(* IEC 61131-3 sources: conversion/test/strings, 10 files *)

(* ---- Asserts.st ---- *)
NAMESPACE AxUnit.Assert

    FUNCTION Equal
        VAR_INPUT
            expected : STRING;
            actual : STRING;
        END_VAR
        Equal(expected := TRUE, actual := expected = actual);
        ;
    END_FUNCTION

END_NAMESPACE

(* ---- ArrayToStringTest.st ---- *)
USING AxUnit.Assert;
USING System.Strings;

NAMESPACE Simatic.Ax.Conversion
    {TestFixture}
    CLASS ArrayToStringTest
        VAR PROTECTED
            array_1_10 : ARRAY[1..10] OF CHAR := ['1', '2', '3', '4', '5', '6', '7', '8', '9', '0'];
            array_0_9 : ARRAY[0..9] OF CHAR := ['0', '1', '2', '3', '4', '5', '6', '7', '8', '9'];
            exp_0_9 : STRING := '0123456789';
            exp_1_10 : STRING := '1234567890';
            empty_string : STRING;
            len : DINT;
            long_array : ARRAY[1..1024] OF CHAR;
            long_string : STRING := '12345678901234567890123456789012345678901234567890123456789012345678901234567890123456789012345678901234567890123456789012345678901234567890123456789012345678901234567890123456789012345678901234567890123456789012345678901234567890123456789012345678901234';
        END_VAR

        {Test}
        METHOD PUBLIC LongArrayTest_expect_StringLength_254
            VAR_TEMP
                _str : STRING;
            END_VAR            Strings.ToArray.OfCharCount(str := long_string, arr := long_array);
            // exceed string lenght
            long_array[255] := '5';
            long_array[256] := '6';
            long_array[257] := '7';

            _str := Arrays.ToString(arr := long_array);

            Equal(expected := 254, actual := LengthOf(_str));
            Equal(expected := long_string, actual := _str);

        END_METHOD

        {Test}
        METHOD PUBLIC Test_Array_ToString_End_smaller_than_start_expect_empty_string
            VAR_TEMP
                _str : STRING;
            END_VAR

            _str := Arrays.ToString(arr := array_0_9, startIdx := 9, endIdx := 5);
            Equal(expected := empty_string, actual := _str);
            ;
        END_METHOD

        {Test}
        METHOD PUBLIC Test_Array_ToString_without_indices_and_expect_full_string
            VAR_TEMP
                _str : STRING;
                array_0_9_test : string := '0123456789';
                array_1_10_test : string := '1234567890';
            END_VAR

            _str := Arrays.ToString(arr := array_0_9);
            Equal(expected := 10, actual := LengthOf(_str));
            Equal(expected := TRUE, actual := _str = array_0_9_test);

            _str := Arrays.ToString(arr := array_1_10);
            Equal(expected := 10, actual := LengthOf(_str));
            Equal(expected := TRUE, actual := _str = array_1_10_test);
            ;
        END_METHOD

        {Test}
        METHOD PUBLIC Test_Array_ToString_part_of_array_and_expect_correct_String
            VAR_TEMP
                _str : STRING;
            END_VAR

            _str := Arrays.ToString(arr := array_0_9, startIdx := 0, endIdx := 0);
            exp_0_9 := '0';
            Equal(expected := 1, actual := LengthOf(_str));
            Equal(expected := exp_0_9, actual := _str);

            _str := Arrays.ToString(arr := array_0_9, startIdx := 1, endIdx := 1);
            exp_0_9 := '1';
            Equal(expected := 1, actual := LengthOf(_str));
            Equal(expected := exp_0_9, actual := _str);

            _str := Arrays.ToString(arr := array_0_9, startIdx := 0, endIdx := 3);
            exp_0_9 := '0123';
            Equal(expected := 4, actual := LengthOf(_str));
            Equal(expected := exp_0_9, actual := _str);

            _str := Arrays.ToString(arr := array_0_9, startIdx := 1, endIdx := 5);
            exp_0_9 := '12345';
            Equal(expected := 5, actual := LengthOf(_str));
            Equal(expected := exp_0_9, actual := _str);

            _str := Arrays.ToString(arr := array_1_10, startIdx := 1, endIdx := 5);
            exp_1_10 := '23456';
            Equal(expected := 5, actual := LengthOf(_str));
            Equal(expected := exp_1_10, actual := _str);
            ;
        END_METHOD

        {Test}
        METHOD PUBLIC Test_Array_Invalid_Indices_Expect_empty_Strings
            VAR_TEMP
                _str : STRING;
            END_VAR

            _str := Arrays.ToString(arr := array_1_10, startIdx := 0, endIdx := 11);
            exp_0_9 := '';
            Equal(expected := 0, actual := LengthOf(_str));
            Equal(expected := exp_0_9, actual := _str);
            ;
            _str := Arrays.ToString(arr := array_1_10, startIdx := 0, endIdx := 10);
            exp_0_9 := '';
            Equal(expected := 0, actual := LengthOf(_str));
            Equal(expected := exp_0_9, actual := _str);

            _str := Arrays.ToString(arr := array_1_10, startIdx := -1, endIdx := 10);
            exp_0_9 := '';
            Equal(expected := 0, actual := LengthOf(_str));
            Equal(expected := exp_0_9, actual := _str);
            ;
        END_METHOD
    END_CLASS
END_NAMESPACE

(* ---- StringToAnyTest.st ---- *)
USING AxUnit.Assert;
USING System.Strings;

NAMESPACE Simatic.Ax.Conversion
    {TestFixture}
    CLASS StrinToAnyIntTest
        VAR
            val : LINT;
            val2 : ULINT;
            res : BOOL;
        END_VAR

        {Test}
        METHOD PUBLIC Convert_STRING_0_TO_LINT_0
            res := StringToAnyInt(str := '0', value => val);
            Equal(expected := 0, actual := val);
            Equal(expected := TRUE, actual := res);
        END_METHOD

        {Test}
        METHOD PUBLIC Convert_STRING_0000000000000000_TO_LINT_0
            res := StringToAnyInt(str := '0000000000000000', value => val);
            Equal(expected := 0, actual := val);
            Equal(expected := TRUE, actual := res);
        END_METHOD

        //ToDo after bugfix
        // {Test(str := STRING#'', value := ULINT#0, success :=FALSE)}
        // {Test(str := STRING#'+', value := ULINT#0, success :=FALSE)}
        // {Test(str := STRING#'-', value := ULINT#0, success :=FALSE)}
        // {Test(str := STRING#'0', value := ULINT#0, success :=TRUE)}
        // {Test(str := STRING#'1', value := ULINT#1, success :=TRUE)}
        // {Test(str := STRING#'2', value := ULINT#2, success :=TRUE)}
        // {Test(str := STRING#'3', value := ULINT#3, success :=TRUE)}
        // {Test(str := STRING#'4', value := ULINT#4, success :=TRUE)}
        // {Test(str := STRING#'5', value := ULINT#5, success :=TRUE)}
        // {Test(str := STRING#'6', value := ULINT#6, success :=TRUE)}
        // {Test(str := STRING#'7', value := ULINT#7, success :=TRUE)}
        // {Test(str := STRING#'8', value := ULINT#8, success :=TRUE)}
        // {Test(str := STRING#'9', value := ULINT#9, success :=TRUE)}
        // {Test(str := STRING#'10', value := ULINT#10, success :=TRUE)}
        // {Test(str := STRING#'15', value := ULINT#15, success :=TRUE)}
        // {Test(str := STRING#'18446744073709551600', value := ULINT#18446744073709551600, success :=TRUE)}
        // {Test(str := STRING#'18446744073709551601', value := ULINT#18446744073709551601, success :=TRUE)}
        // {Test(str := STRING#'18446744073709551602', value := ULINT#18446744073709551602, success :=TRUE)}
        // {Test(str := STRING#'18446744073709551603', value := ULINT#18446744073709551603, success :=TRUE)}
        // {Test(str := STRING#'18446744073709551604', value := ULINT#18446744073709551604, success :=TRUE)}
        // {Test(str := STRING#'18446744073709551605', value := ULINT#18446744073709551605, success :=TRUE)}
        // {Test(str := STRING#'18446744073709551606', value := ULINT#18446744073709551606, success :=TRUE)}
        // {Test(str := STRING#'18446744073709551607', value := ULINT#18446744073709551607, success :=TRUE)}
        // {Test(str := STRING#'18446744073709551608', value := ULINT#18446744073709551608, success :=TRUE)}
        // {Test(str := STRING#'18446744073709551609', value := ULINT#18446744073709551609, success :=TRUE)}
        // {Test(str := STRING#'18446744073709551610', value := ULINT#18446744073709551610, success :=TRUE)}
        // {Test(str := STRING#'18446744073709551611', value := ULINT#18446744073709551611, success :=TRUE)}
        // {Test(str := STRING#'18446744073709551612', value := ULINT#18446744073709551612, success :=TRUE)}
        // {Test(str := STRING#'18446744073709551613', value := ULINT#18446744073709551613, success :=TRUE)}
        // {Test(str := STRING#'18446744073709551614', value := ULINT#18446744073709551614, success :=TRUE)}
        // {Test(str := STRING#'18446744073709551615', value := ULINT#18446744073709551615, success :=TRUE)}
        // {Test(str := STRING#'18446744073709551616', value := ULINT#0, success :=FALSE)}
        // {Test(str := STRING#'18446744073709551617', value := ULINT#0, success :=FALSE)}
        // {Test(str := STRING#'18446744073709551618', value := ULINT#0, success :=FALSE)}
        // {Test(str := STRING#'18446744073709551619', value := ULINT#0, success :=FALSE)}
        // {Test(str := STRING#'18446744073709551620', value := ULINT#0, success :=FALSE)}
        // {Test(str := STRING#'18446744073709551621', value := ULINT#0, success :=FALSE)}
        // {Test(str := STRING#'18446744073709551622', value := ULINT#0, success :=FALSE)}
        // {Test(str := STRING#'18446744073709551623', value := ULINT#0, success :=FALSE)}
        // {Test(str := STRING#'18446744073709551624', value := ULINT#0, success :=FALSE)}
        // {Test(str := STRING#'18446744073709551625', value := ULINT#0, success :=FALSE)}
        // {Test(str := STRING#'18446744073709551626', value := ULINT#0, success :=FALSE)}
        // {Test(str := STRING#'18446744073709551636', value := ULINT#0, success :=FALSE)}
        // {Test(str := STRING#'18446744073709551746', value := ULINT#0, success :=FALSE)}
        // {Test(str := STRING#'18446744073709551800', value := ULINT#0, success :=FALSE)}
        // {Test(str := STRING#'20000000000000000000', value := ULINT#0, success :=FALSE)}
        // METHOD PUBLIC Convert_STRING_TO_ULINT
        //     VAR_INPUT
        //         str : STRING;
        //         value : ULINT;
        //         success : BOOL;
        //     END_VAR
        //     VAR_TEMP
        //         resVal : ULINT;
        //     END_VAR
        //     res := StringToULint(str := str, value => resVal);
        //     Equal(expected := value, actual := resVal);
        //     Equal(expected := success, actual := res);
        // END_METHOD

        // {Test(str := STRING#'', value := LINT#0, success :=FALSE)}
        // {Test(str := STRING#'+', value := LINT#0, success :=FALSE)}
        // {Test(str := STRING#'-', value := LINT#0, success :=FALSE)}
        // {Test(str := STRING#'0', value := LINT#0, success :=TRUE)}
        // {Test(str := STRING#'1', value := LINT#1, success :=TRUE)}
        // {Test(str := STRING#'2', value := LINT#2, success :=TRUE)}
        // {Test(str := STRING#'3', value := LINT#3, success :=TRUE)}
        // {Test(str := STRING#'4', value := LINT#4, success :=TRUE)}
        // {Test(str := STRING#'5', value := LINT#5, success :=TRUE)}
        // {Test(str := STRING#'6', value := LINT#6, success :=TRUE)}
        // {Test(str := STRING#'7', value := LINT#7, success :=TRUE)}
        // {Test(str := STRING#'8', value := LINT#8, success :=TRUE)}
        // {Test(str := STRING#'9', value := LINT#9, success :=TRUE)}
        // {Test(str := STRING#'10', value := LINT#10, success :=TRUE)}
        // {Test(str := STRING#'15', value := LINT#15, success :=TRUE)}
        // {Test(str := STRING#'-0', value := LINT#0, success :=TRUE)}
        // {Test(str := STRING#'-1', value := LINT#-1, success :=TRUE)}
        // {Test(str := STRING#'-2', value := LINT#-2, success :=TRUE)}
        // {Test(str := STRING#'-3', value := LINT#-3, success :=TRUE)}
        // {Test(str := STRING#'-4', value := LINT#-4, success :=TRUE)}
        // {Test(str := STRING#'-5', value := LINT#-5, success :=TRUE)}
        // {Test(str := STRING#'-6', value := LINT#-6, success :=TRUE)}
        // {Test(str := STRING#'-7', value := LINT#-7, success :=TRUE)}
        // {Test(str := STRING#'-8', value := LINT#-8, success :=TRUE)}
        // {Test(str := STRING#'-9', value := LINT#-9, success :=TRUE)}
        // {Test(str := STRING#'-10', value := LINT#-10, success :=TRUE)}
        // {Test(str := STRING#'-15', value := LINT#-15, success :=TRUE)}
        // {Test(str := STRING#'9223372036854775799', value := LINT#9223372036854775799, success :=TRUE)}
        // {Test(str := STRING#'9223372036854775800', value := LINT#9223372036854775800, success :=TRUE)}
        // {Test(str := STRING#'9223372036854775801', value := LINT#9223372036854775801, success :=TRUE)}
        // {Test(str := STRING#'9223372036854775802', value := LINT#9223372036854775802, success :=TRUE)}
        // {Test(str := STRING#'9223372036854775803', value := LINT#9223372036854775803, success :=TRUE)}
        // {Test(str := STRING#'9223372036854775804', value := LINT#9223372036854775804, success :=TRUE)}
        // {Test(str := STRING#'9223372036854775805', value := LINT#9223372036854775805, success :=TRUE)}
        // {Test(str := STRING#'9223372036854775806', value := LINT#9223372036854775806, success :=TRUE)}
        // {Test(str := STRING#'9223372036854775807', value := LINT#9223372036854775807, success :=TRUE)}
        // {Test(str := STRING#'9223372036854775808', value := LINT#0, success :=FALSE)}
        // {Test(str := STRING#'9223372036854775809', value := LINT#0, success :=FALSE)}
        // {Test(str := STRING#'9223372036854775810', value := LINT#0, success :=FALSE)}
        // {Test(str := STRING#'9223372036854775811', value := LINT#0, success :=FALSE)}
        // {Test(str := STRING#'19223372036854775811', value := LINT#0, success :=FALSE)}

        // {Test(str := STRING#'-9223372036854775799', value := LINT#-9223372036854775799, success :=TRUE)}
        // {Test(str := STRING#'-9223372036854775800', value := LINT#-9223372036854775800, success :=TRUE)}
        // {Test(str := STRING#'-9223372036854775801', value := LINT#-9223372036854775801, success :=TRUE)}
        // {Test(str := STRING#'-9223372036854775802', value := LINT#-9223372036854775802, success :=TRUE)}
        // {Test(str := STRING#'-9223372036854775803', value := LINT#-9223372036854775803, success :=TRUE)}
        // {Test(str := STRING#'-9223372036854775804', value := LINT#-9223372036854775804, success :=TRUE)}
        // {Test(str := STRING#'-9223372036854775805', value := LINT#-9223372036854775805, success :=TRUE)}
        // {Test(str := STRING#'-9223372036854775806', value := LINT#-9223372036854775806, success :=TRUE)}
        // {Test(str := STRING#'-9223372036854775807', value := LINT#-9223372036854775807, success :=TRUE)}
        // {Test(str := STRING#'-9223372036854775808', value := LINT#-9223372036854775808, success :=TRUE)}
        // {Test(str := STRING#'-9223372036854775809', value := LINT#0, success :=FALSE)}
        // {Test(str := STRING#'-9223372036854775810', value := LINT#0, success :=FALSE)}
        // {Test(str := STRING#'-9223372036854775811', value := LINT#0, success :=FALSE)}
        // {Test(str := STRING#'-19223372036854775811', value := LINT#0, success :=FALSE)}
        // METHOD PUBLIC Convert_STRING_TO_ANYINT
        //     VAR_INPUT
        //         str : STRING;
        //         value : LINT;
        //         success : BOOL;
        //     END_VAR
        //     VAR_TEMP
        //         resVal : LINT;
        //     END_VAR
        //     res := StringToAnyInt(str := str, value => resVal);
        //     Equal(expected := value, actual := resVal);
        //     Equal(expected := success, actual := res);
        // END_METHOD

        {Test}
        METHOD PUBLIC Convert_STRING_123_TO_LINT_123
            res := StringToAnyInt(str := '123', value => val);
            Equal(expected := 123, actual := val);
            Equal(expected := TRUE, actual := res);
        END_METHOD

        {Test}
        METHOD PUBLIC Convert_STRING_00000000123_TO_LINT_123
            res := StringToAnyInt(str := '123', value => val);
            Equal(expected := 123, actual := val);
            Equal(expected := TRUE, actual := res);
        END_METHOD

        {Test}
        METHOD PUBLIC Convert_STRING_PLUS_123_TO_LINT_123
            res := StringToAnyInt(str := '+00000000123', value => val);
            Equal(expected := 123, actual := val);
            Equal(expected := TRUE, actual := res);
        END_METHOD

        {Test}
        METHOD PUBLIC Convert_STRING_MINUS_0000000000123_TO_LINT_123
            res := StringToAnyInt(str := '-00000000123', value => val);
            Equal(expected := -123, actual := val);
            Equal(expected := TRUE, actual := res);
        END_METHOD

        {Test}
        METHOD PUBLIC Convert_STRING_MINUS_123_TO_LINT_123
            res := StringToAnyInt(str := '-123', value => val);
            Equal(expected := -123, actual := val);
            Equal(expected := TRUE, actual := res);
        END_METHOD

        {Test}
        METHOD PUBLIC Convert_STRING_MINUS_1234567890_TO_LINT_1234567890
            res := StringToAnyInt(str := '-1234567890', value => val);
            Equal(expected := LINT#-1234567890, actual := val);
            Equal(expected := TRUE, actual := res);
        END_METHOD

        {Test}
        METHOD PUBLIC Convert_STRING_9223372036854775807_TO_LINT_9223372036854775807
            res := StringToAnyInt(str := '9223372036854775807', value => val);
            Equal(expected := LINT#9223372036854775807, actual := val);
            Equal(expected := TRUE, actual := res);
            res := StringToAnyInt(str := '+9223372036854775807', value => val);
            Equal(expected := LINT#9223372036854775807, actual := val);
            Equal(expected := TRUE, actual := res);

        END_METHOD

        {Test}
        METHOD PUBLIC Convert_STRING_MINUS_9223372036854775808_TO_LINT_9223372036854775808
            res := StringToAnyInt(str := '-9223372036854775808', value => val);
            Equal(expected := LINT#-9223372036854775808, actual := val);
            Equal(expected := TRUE, actual := res);
        END_METHOD

        {Test}
        METHOD PUBLIC Convert_STRING_18446744073709551615_TO_ULINT_18446744073709551615
            res := StringToULINT(str := '18446744073709551615', value => val2);
            Equal(expected := ULINT#18446744073709551615, actual := val2);
            Equal(expected := TRUE, actual := res);

            res := StringToULINT(str := '+18446744073709551615', value => val2);
            Equal(expected := ULINT#18446744073709551615, actual := val2);
            Equal(expected := TRUE, actual := res);
        END_METHOD

        {Test}
        METHOD PUBLIC Convert_WrongStrings_ExpectFalse
            res := StringToAnyInt(str := '+-123', value => val);
            Equal(expected := 0, actual := val);
            Equal(expected := FALSE, actual := res);

            res := StringToAnyInt(str := '000+123', value => val);
            Equal(expected := 0, actual := val);
            Equal(expected := FALSE, actual := res);

            res := StringToAnyInt(str := '1000+123', value => val);
            Equal(expected := 0, actual := val);
            Equal(expected := FALSE, actual := res);

            res := StringToAnyInt(str := 'aaa', value => val);
            Equal(expected := 0, actual := val);
            Equal(expected := FALSE, actual := res);

            res := StringToAnyInt(str := '12a23', value => val);
            Equal(expected := 0, actual := val);
            Equal(expected := FALSE, actual := res);

        END_METHOD
    END_CLASS
END_NAMESPACE

(* ---- StringToArrayOfLintCountTest.st ---- *)
USING AxUnit.Assert;
USING System.Strings;

NAMESPACE Simatic.Ax.Conversion.Strings.ToArray
    {TestFixture}
    CLASS StringToArrayOfLIntCountTest
        VAR
            arr: ARRAY[0..3] OF LINT;
        END_VAR

        {Test}
        METHOD PUBLIC EmptyArray_ReturnsFalse
            VAR
                str: STRING := '';
                count: DINT;
            END_VAR

            count := ToArray.OfLintCount(str, arr);
            Equal(0, count);

            str:= '   ';
            count := ToArray.OfLintCount(str, arr);
            Equal(0, count);
        END_METHOD

        {Test}
        METHOD PUBLIC NotArray_ReturnsFalse
            VAR
                str: STRING := 'hello';
                count: DINT;
            END_VAR
            count := ToArray.OfLintCount(str, arr);
            Equal(0, count);
        END_METHOD

        {Test}
        METHOD PUBLIC WrongArray_ReturnsFalse
            VAR
                str: STRING := '["hello", "goodbye"]';
                count: DINT;
            END_VAR
            count := ToArray.OfLintCount(str, arr);
            Equal(0, count);
        END_METHOD

        {Test}
        METHOD PUBLIC Array_Converts
            VAR
                str: STRING := '[12, 345, 6789, 101112]';
                count: DINT;
            END_VAR
            count := ToArray.OfLintCount(str, arr);
            Equal(4, count);
            Equal(LINT#12, arr[0]);
            Equal(LINT#345, arr[1]);
            Equal(LINT#6789, arr[2]);
            Equal(LINT#101112, arr[3]);
        END_METHOD

        {Test}
        METHOD PUBLIC Array_Converts_with_spaces
            VAR
                str: STRING := '   [   12,   345   ,    6789    ,    101112    ]   ';
                count: DINT;
            END_VAR
            count := ToArray.OfLintCount(str, arr);
            Equal(4, count);
            Equal(LINT#12, arr[0]);
            Equal(LINT#345, arr[1]);
            Equal(LINT#6789, arr[2]);
            Equal(LINT#101112, arr[3]);
        END_METHOD

        {Test}
        METHOD PUBLIC Smaller_Array_Converts_with_spaces
            VAR
                str: STRING := '   [   345   ,    6789    ,    101112    ]   ';
                count: DINT;
            END_VAR
            count := ToArray.OfLintCount(str, arr);
            Equal(3, count);
            Equal(LINT#345, arr[0]);
            Equal(LINT#6789, arr[1]);
            Equal(LINT#101112, arr[2]);
        END_METHOD

        {Test}
        METHOD PUBLIC Array_Converts_toSmallArray
            VAR
                str: STRING := '[12, 345, 6789, 101112, 1234]';
                count: DINT;
            END_VAR
            count := ToArray.OfLintCount(str, arr);
            Equal(4, count);
            Equal(LINT#12, arr[0]);
            Equal(LINT#345, arr[1]);
            Equal(LINT#6789, arr[2]);
            Equal(LINT#101112, arr[3]);
        END_METHOD

        {Test}
        METHOD PUBLIC Array_Converts_toBigArray
            VAR
                str: STRING := '[12, 345, 6789]';
                count: DINT;
            END_VAR
            count := ToArray.OfLintCount(str, arr);
            Equal(3, count);
            Equal(LINT#12, arr[0]);
            Equal(LINT#345, arr[1]);
            Equal(LINT#6789, arr[2]);
        END_METHOD

    END_CLASS
END_NAMESPACE

(* ---- StringToArrayTest.st ---- *)
USING AxUnit.Assert;
USING System.Strings;

NAMESPACE Simatic.Ax.Conversion
    {TestFixture}
    CLASS StrinToArrayIntTest
        VAR PROTECTED
            s10 : STRING := '0123456789';
            s16 : STRING := '0123456789ABCDEF';
            a0_9 : ARRAY[0..9] OF CHAR;
            a10_19 : ARRAY[10..19] OF CHAR;

            a0_12 : ARRAY[0..12] OF CHAR;
            a10_22 : ARRAY[10..12] OF CHAR;
            len : DINT;
        END_VAR

        {Test}
        METHOD PUBLIC Test_array_and_string_length_is_equal_expect_lenght_10
            len := Strings.ToArray.OfCharCount(s10, a0_9);
            Equal(expected := 10, actual := len);
            Equal(expected := '0', actual := a0_9[0]);
            Equal(expected := '1', actual := a0_9[1]);
            Equal(expected := '8', actual := a0_9[8]);
            Equal(expected := '9', actual := a0_9[9]);
        END_METHOD

        {Test}
        METHOD PUBLIC Test_array_starting_with_10_and_string_length_is_equal_expect_lenght_10
            len := Strings.ToArray.OfCharCount(s10, a10_19);
            Equal(expected := 10, actual := len);
            Equal(expected := '0', actual := a10_19[10]);
            Equal(expected := '1', actual := a10_19[11]);
            Equal(expected := '8', actual := a10_19[18]);
            Equal(expected := '9', actual := a10_19[19]);
        END_METHOD

        {Test}
        METHOD PUBLIC Test_array_and_string_length_is_longer_expect_lenght_10
            len := Strings.ToArray.OfCharCount(s16, a0_9);
            Equal(expected := 10, actual := len);
            Equal(expected := '0', actual := a0_9[0]);
            Equal(expected := '1', actual := a0_9[1]);
            Equal(expected := '8', actual := a0_9[8]);
            Equal(expected := '9', actual := a0_9[9]);
        END_METHOD

        {Test}
        METHOD PUBLIC Test_array_starting_with_10_and_string_length_is_longer_expect_lenght_10
            len := Strings.ToArray.OfCharCount(s16, a10_19);
            Equal(expected := 10, actual := len);
            Equal(expected := '0', actual := a10_19[10]);
            Equal(expected := '1', actual := a10_19[11]);
            Equal(expected := '8', actual := a10_19[18]);
            Equal(expected := '9', actual := a10_19[19]);
        END_METHOD

        {Test}
        METHOD PUBLIC Test_array_and_string_length_buffer_is_longer_expect_lenght_10
            len := Strings.ToArray.OfCharCount(s10, a0_12);
            Equal(expected := 10, actual := len);
            Equal(expected := '0', actual := a0_12[0]);
            Equal(expected := '1', actual := a0_12[1]);
            Equal(expected := '8', actual := a0_12[8]);
            Equal(expected := '9', actual := a0_12[9]);
            Equal(expected := TO_CHAR(BYTE#0), actual := a0_12[10]);
            Equal(expected := TO_CHAR(BYTE#0), actual := a0_12[11]);
            Equal(expected := TO_CHAR(BYTE#0), actual := a0_12[12]);

            len := Strings.ToArray.OfCharCount(s16, a0_12);
            Equal(expected := 13, actual := len);
        END_METHOD

        {Test}
        METHOD PUBLIC Test_array_and_string_length_buffer_is_shorter_expect_lenght_13

            len := Strings.ToArray.OfCharCount(s16, a0_12);
            Equal(expected := 13, actual := len);
            Equal(expected := '0', actual := a0_12[0]);
            Equal(expected := '1', actual := a0_12[1]);
            Equal(expected := '8', actual := a0_12[8]);
            Equal(expected := '9', actual := a0_12[9]);
            Equal(expected := 'A', actual := a0_12[10]);
            Equal(expected := 'B', actual := a0_12[11]);
            Equal(expected := 'C', actual := a0_12[12]);
        END_METHOD
    END_CLASS
END_NAMESPACE

(* ---- TestDifferentTypeConversions.st ---- *)
USING AxUnit.Assert;
using System.Strings;

NAMESPACE Simatic.Ax.Conversion
    {TestFixture}
    CLASS TestDifferentTypeConversions
        {Test}
        METHOD PUBLIC Test_SINT
            Equal(expected := '0', actual := Integer.ToString(value := SINT#0));
            Equal(expected := '127', actual := Integer.ToString(value := SINT#127));
            Equal(expected := '+127', actual := Integer.ToString(value := USINT#127, mode := ConversionMode#FORCE_SIGN));
            Equal(expected := '-128', actual := Integer.ToString(value := SINT#-128));
        END_METHOD

        {Test}
        METHOD PUBLIC Test_USINT
            Equal(expected := '0', actual := Integer.ToString(value := USINT#0));
            Equal(expected := '255', actual := Integer.ToString(value := USINT#255));
            Equal(expected := '+255', actual := Integer.ToString(value := USINT#255, mode := ConversionMode#FORCE_SIGN));
        END_METHOD

        {Test}
        METHOD PUBLIC Test_INT
            Equal(expected := '0', actual := Integer.ToString(value := INT#0));
            Equal(expected := '32767', actual := Integer.ToString(value := INT#32767));
            Equal(expected := '+32767', actual := Integer.ToString(value := INT#32767, mode := ConversionMode#FORCE_SIGN));
            Equal(expected := '-32768', actual := Integer.ToString(value := INT#-32768));

        END_METHOD

        {Test}
        METHOD PUBLIC Test_UINT
            Equal(expected := '0', actual := Integer.ToString(value := UINT#0));
            Equal(expected := '65535', actual := Integer.ToString(value := UINT#65535));
            Equal(expected := '+65535', actual := Integer.ToString(value := UINT#65535, mode := ConversionMode#FORCE_SIGN));

        END_METHOD

        {Test}
        METHOD PUBLIC Test_DINT
            Equal(expected := '0', actual := Integer.ToString(value := DINT#0));
            Equal(expected := '2147483647', actual := Integer.ToString(value := DINT#2147483647));
            Equal(expected := '+2147483647', actual := Integer.ToString(value := UDINT#2147483647, mode := ConversionMode#FORCE_SIGN));
            Equal(expected := '-2147483648', actual := Integer.ToString(value := DINT#-2147483648));
        END_METHOD

        {Test}
        METHOD PUBLIC Test_UDINT
            Equal(expected := '0', actual := Integer.ToString(value := UDINT#0));
            Equal(expected := '+4294967295', actual := Integer.ToString(value := UDINT#4294967295, mode := ConversionMode#FORCE_SIGN));
            Equal(expected := '4294967295', actual := Integer.ToString(value := UDINT#4294967295));
        END_METHOD

        {Test}
        METHOD PUBLIC Test_LINT
            Equal(expected := '0', actual := Integer.ToString(value := DINT#0));
            Equal(expected := '9223372036854775807', actual := Integer.ToString(value := LINT#9223372036854775807));
            Equal(expected := '+9223372036854775807', actual := Integer.ToString(value := LINT#9223372036854775807, mode := ConversionMode#FORCE_SIGN));
            Equal(expected := '-9223372036854775808', actual := Integer.ToString(value := LINT#-9223372036854775808));
        END_METHOD

        {Test}
        METHOD PUBLIC Test_ULINT
            Equal(expected := '0', actual := Integer.ToString(value := UDINT#0));
            Equal(expected := '18446744073709551615', actual := Integer.ToString(value := ULINT#18446744073709551615));
            Equal(expected := '+18446744073709551615', actual := Integer.ToString(value := ULINT#18446744073709551615, mode := ConversionMode#FORCE_SIGN));

        END_METHOD

    END_CLASS
END_NAMESPACE

(* ---- TestGetHexValueOfChar.st ---- *)
USING AxUnit.Assert;
NAMESPACE Simatic.Ax.Conversion
    {TestFixture}
    CLASS TestGetHexValueOfChar
        VAR PROTECTED
            res : BYTE;
            ret : bool;
        END_VAR

        {Test(c := 'a', n := 1, exp := BYTE#16#a)}
        {Test(c := 'b', n := 1, exp := BYTE#16#b)}
        {Test(c := 'c', n := 1, exp := BYTE#16#c)}
        {Test(c := 'd', n := 1, exp := BYTE#16#d)}
        {Test(c := 'e', n := 1, exp := BYTE#16#e)}
        {Test(c := 'f', n := 1, exp := BYTE#16#f)}
        {Test(c := 'A', n := 1, exp := BYTE#16#a)}
        {Test(c := 'B', n := 1, exp := BYTE#16#b)}
        {Test(c := 'C', n := 1, exp := BYTE#16#c)}
        {Test(c := 'D', n := 1, exp := BYTE#16#d)}
        {Test(c := 'E', n := 1, exp := BYTE#16#e)}
        {Test(c := 'F', n := 1, exp := BYTE#16#f)}
        {Test(c := '0', n := 1, exp := BYTE#16#0)}
        {Test(c := '1', n := 1, exp := BYTE#16#1)}
        {Test(c := '2', n := 1, exp := BYTE#16#2)}
        {Test(c := '3', n := 1, exp := BYTE#16#3)}
        {Test(c := '4', n := 1, exp := BYTE#16#4)}
        {Test(c := '5', n := 1, exp := BYTE#16#5)}
        {Test(c := '6', n := 1, exp := BYTE#16#6)}
        {Test(c := '7', n := 1, exp := BYTE#16#7)}
        {Test(c := '8', n := 1, exp := BYTE#16#8)}
        {Test(c := '9', n := 1, exp := BYTE#16#9)}
        METHOD PUBLIC ConvertHexCharsToByteValue
            VAR_INPUT
                c : CHAR;
                n : INT;
                exp : BYTE;
            END_VAR
            ret := GetHexValueOfChar(c := c, result => res);
            Equal(expected := exp, actual := res);
            Equal(expected := TRUE, actual := ret);
            ;
        END_METHOD

        {Test}
        METHOD PUBLIC InvalidCharacter
            ret := GetHexValueOfChar(c := 'h', result => res);
            Equal(expected := FALSE, actual := ret);
        END_METHOD
    END_CLASS
END_NAMESPACE

(* ---- TestStringToHex.st ---- *)
USING AxUnit.Assert;
NAMESPACE Simatic.Ax.Conversion.Strings
    {TestFixture}
    CLASS TestStringToHex
        VAR PROTECTED
            res : DWORD;
            ret : WORD;
        END_VAR

        //ToDo after bugfix
        // {Test(str := 'a', n := 1, exp := DWORD#16#a)}
        // {Test(str := 'b', n := 1, exp := DWORD#16#b)}
        // {Test(str := 'c', n := 1, exp := DWORD#16#c)}
        // {Test(str := 'd', n := 1, exp := DWORD#16#d)}
        // {Test(str := 'e', n := 1, exp := DWORD#16#e)}
        // {Test(str := 'f', n := 1, exp := DWORD#16#f)}
        // {Test(str := 'A', n := 1, exp := DWORD#16#a)}
        // {Test(str := 'B', n := 1, exp := DWORD#16#b)}
        // {Test(str := 'C', n := 1, exp := DWORD#16#c)}
        // {Test(str := 'D', n := 1, exp := DWORD#16#d)}
        // {Test(str := 'E', n := 1, exp := DWORD#16#e)}
        // {Test(str := 'F', n := 1, exp := DWORD#16#f)}
        // {Test(str := '0', n := 1, exp := DWORD#16#0)}
        // {Test(str := '1', n := 1, exp := DWORD#16#1)}
        // {Test(str := '2', n := 1, exp := DWORD#16#2)}
        // {Test(str := '3', n := 1, exp := DWORD#16#3)}
        // {Test(str := '4', n := 1, exp := DWORD#16#4)}
        // {Test(str := '5', n := 1, exp := DWORD#16#5)}
        // {Test(str := '6', n := 1, exp := DWORD#16#6)}
        // {Test(str := '7', n := 1, exp := DWORD#16#7)}
        // {Test(str := '8', n := 1, exp := DWORD#16#8)}
        // {Test(str := '9', n := 1, exp := DWORD#16#9)}
        // {Test(str := 'aFFe', n := 4, exp := DWORD#16#affe)}
        // {Test(str := 'aa', n := 2, exp := DWORD#16#aa)}
        // {Test(str := '12', n := 2, exp := DWORD#16#12)}
        // {Test(str := '123', n := 3, exp := DWORD#16#123)}
        // {Test(str := '1234', n := 4, exp := DWORD#16#1234)}
        // METHOD PUBLIC ConvertDifferentValidStringsToDWORD
        //     VAR_INPUT
        //         str : STRING;
        //         n : INT;
        //         exp : DWORD;
        //     END_VAR
        //     ret := ToHex(str := str, n := n, result => res);
        //     Equal(expected := exp, actual := res);
        //     Equal(expected := WORD#16#0000, actual := ret);
        //     ;
        // END_METHOD

        {Test}
        METHOD PUBLIC InvalidCharacter
            ret := ToHex(str := 'afgh', n := 4, result => res);
            Equal(expected := WORD#16#0007, actual := ret);
        END_METHOD

        {Test}
        METHOD PUBLIC InputSmallerThanN
            ret := ToHex(str := 'af', n := 3, result => res);
            Equal(expected := WORD#16#8182, actual := ret);
        END_METHOD

        {Test}
        METHOD PUBLIC OutputBufferToSmall
            ret := ToHex(str := '1234567890', n := 10, result => res);
            Equal(expected := WORD#16#8482, actual := ret);
        END_METHOD
    END_CLASS
END_NAMESPACE

(* ---- ToStringTest.st ---- *)
USING AxUnit.Assert;
USING System.Strings;

NAMESPACE Simatic.Ax.Conversion
    {TestFixture}
    CLASS ToStringTest
        VAR
            s : STRING;
        END_VAR
        {Test}
        METHOD PUBLIC Convert_INT_1234_ToString_Expect_1234
            s := AnyIntToString(value := 1234);
            Equal(expected := '1234', actual := s);
            Equal(expected := 4, actual := LengthOf(s));
        END_METHOD

        {Test}
        METHOD PUBLIC Convert_INT_MINUS_1234_ToString_Expect_MINUS_1234
            s := AnyIntToString(value := -1234);
            Equal(expected := '-1234', actual := s);
            Equal(expected := 5, actual := LengthOf(s));
        END_METHOD

        {Test}
        METHOD PUBLIC Convert_INT_VALUES_ToString_Expect_Value_AsString
            // 0
            s := AnyIntToString(value := 0);
            Equal(expected := '0', actual := s);
            Equal(expected := 1, actual := LengthOf(s));

            // 1
            s := AnyIntToString(value := 1);
            Equal(expected := '1', actual := s);
            Equal(expected := 1, actual := LengthOf(s));

            // 1
            s := AnyIntToString(value := -1);
            Equal(expected := '-1', actual := s);
            Equal(expected := 2, actual := LengthOf(s));

            // 99
            s := AnyIntToString(value := 99);
            Equal(expected := '99', actual := s);
            Equal(expected := 2, actual := LengthOf(s));

            // -99
            s := AnyIntToString(value := -99);
            Equal(expected := '-99', actual := s);
            Equal(expected := 3, actual := LengthOf(s));

            // 1234567890
            s := AnyIntToString(value := DINT#1234567890);
            Equal(expected := '1234567890', actual := s);
            Equal(expected := 10, actual := LengthOf(s));

            // -1234567890
            s := AnyIntToString(value := DINT#-1234567890);
            Equal(expected := '-1234567890', actual := s);
            Equal(expected := 11, actual := LengthOf(s));

            // 9223372036854775807
            s := AnyIntToString(value := LINT#9223372036854775807);
            Equal(expected := '9223372036854775807', actual := s);
            Equal(expected := 19, actual := LengthOf(s));

            // -9223372036854775808
            s := AnyIntToString(value := LINT#-9223372036854775808);
            Equal(expected := '-9223372036854775808', actual := s);
            Equal(expected := 20, actual := LengthOf(s));

            // -9223372036854775808
            s := ULintToString(value := ULINT#18446744073709551615);
            Equal(expected := '18446744073709551615', actual := s);
            Equal(expected := 20, actual := LengthOf(s));

        END_METHOD

        {Test}
        METHOD PUBLIC Convert_Integers_with_forced_sign
            // 0
            s := AnyIntToString(value := 0, mode := ConversionMode#FORCE_SIGN);
            Equal(expected := '0', actual := s);
            Equal(expected := 1, actual := LengthOf(s));

            // 1
            s := AnyIntToString(value := 1, mode := ConversionMode#FORCE_SIGN);
            Equal(expected := '+1', actual := s);
            Equal(expected := 2, actual := LengthOf(s));

            // 1
            s := AnyIntToString(value := -1, mode := ConversionMode#FORCE_SIGN);
            Equal(expected := '-1', actual := s);
            Equal(expected := 2, actual := LengthOf(s));

            // 99
            s := AnyIntToString(value := 99, mode := ConversionMode#FORCE_SIGN);
            Equal(expected := '+99', actual := s);
            Equal(expected := 3, actual := LengthOf(s));

            // -99
            s := AnyIntToString(value := -99, mode := ConversionMode#FORCE_SIGN);
            Equal(expected := '-99', actual := s);
            Equal(expected := 3, actual := LengthOf(s));

            // 9223372036854775807
            s := AnyIntToString(value := LINT#9223372036854775807, mode := ConversionMode#FORCE_SIGN);
            Equal(expected := '+9223372036854775807', actual := s);
            Equal(expected := 20, actual := LengthOf(s));

            // -9223372036854775808
            s := AnyIntToString(value := LINT#-9223372036854775808, mode := ConversionMode#FORCE_SIGN);
            Equal(expected := '-9223372036854775808', actual := s);
            Equal(expected := 20, actual := LengthOf(s));
        END_METHOD

        //ToDo after bugfix
        // Blocked by HA-1737
        // {Test(v := 1234, expStr := '1234', len := 4)}
        // METHOD PUBLIC Convert_INT_VALUES_ToString_Expect_Value_AsString2
        //     VAR_INPUT
        //         v : LINT;
        //         expStr : STRING;
        //         len : INT;
        //     END_VAR
        //     ;
        //     s := Integer.ToString(value := v);
        //     Equal(expected := expStr, actual := s);
        //     Equal(expected := len, actual := LengthOf(s));
        // END_METHOD

    END_CLASS
END_NAMESPACE

(* ---- HexToString.st ---- *)
USING AxUnit.Assert;
USING System.Strings;

NAMESPACE Simatic.Ax.Conversion
    // {TestFixture}
    // CLASS HexToString

    //ToDo after bugfix
    //     {Test (b:= BYTE#16#00, hex := STRING#'00')}
    //     {Test (b:= BYTE#16#11, hex := STRING#'11')}
    //     {Test (b:= BYTE#16#22, hex := STRING#'22')}
    //     {Test (b:= BYTE#16#33, hex := STRING#'33')}
    //     {Test (b:= BYTE#16#44, hex := STRING#'44')}
    //     {Test (b:= BYTE#16#55, hex := STRING#'55')}
    //     {Test (b:= BYTE#16#66, hex := STRING#'66')}
    //     {Test (b:= BYTE#16#77, hex := STRING#'77')}
    //     {Test (b:= BYTE#16#88, hex := STRING#'88')}
    //     {Test (b:= BYTE#16#99, hex := STRING#'99')}
    //     {Test (b:= BYTE#16#AA, hex := STRING#'AA')}
    //     {Test (b:= BYTE#16#BB, hex := STRING#'BB')}
    //     {Test (b:= BYTE#16#CC, hex := STRING#'CC')}
    //     {Test (b:= BYTE#16#DD, hex := STRING#'DD')}
    //     {Test (b:= BYTE#16#EE, hex := STRING#'EE')}
    //     {Test (b:= BYTE#16#FF, hex := STRING#'FF')}

    //     METHOD PUBLIC Convert_Hex_Byte_To_String

    //         VAR_INPUT
    //             b : BYTE;
    //             hex : STRING;
    //         END_VAR
    //         VAR_TEMP
    //             s : STRING;
    //         END_VAR

    //         s := ByteToString(b);
    //         Equal(expected := hex, actual := s);

    //     END_METHOD

    // END_CLASS
END_NAMESPACE
